(* IEC 61131-3 sources: programs/VI-54/VI-54_20171205/VI-54_20171205/Stations/Screen/LseClass170718/Class/CalcDeltaSC, 1 file *)

(* ---- CalcDeltaSC.st ---- *)
(*!
<Class
	Name               = "CalcDeltaSC"
	Revision           = "0.0"
	RealtimeTask       = "false"
	CyclicTask         = "false"
	BackgroundTask     = "false"
	Sigmatek           = "false"
	OSInterface        = "false"
	HighPriority       = "false"
	Automatic          = "false"
	UpdateMode         = "Prescan"
	SharedCommandTable = "true"
	Objectsize         = "(450,1320)">
	<Channels>
		<Server Name="OffsetZ" Visualized="false" Initialize="false" WriteProtected="false" Retentive="false"/>
	</Channels>
	<Network Name="CalcDeltaSC">
		<!-- List of Components in this network -->
		<Components>
			<Object
				Name       = "_base"
				Class      = "CalcDelta"
				Position   = "(218,120)"
				Visualized = "true"
				Remotely   = "true">
				<Channels>
					<Server Name="ActPos1"/>
					<Server Name="ActPos2"/>
					<Server Name="ActPos3"/>
					<Server Name="ActPos4"/>
					<Server Name="ClassSvr"/>
					<Server Name="DragCalcDelay" Value="0"/>
					<Server Name="HeadRadius" Value="500000"/>
					<Server Name="MotorArm" Value="3200000"/>
					<Server Name="MotorRadius" Value="2000000"/>
					<Server Name="RobotArm" Value="8500000"/>
					<Server Name="RobotRotAxisZ"/>
					<Server Name="SetPos1_Control"/>
					<Server Name="SetPos2_Control"/>
					<Server Name="SetPos3_Control"/>
					<Server Name="SetPos4_Control"/>
					<Server Name="XW1"/>
					<Server Name="XW2"/>
					<Server Name="XW3"/>
					<Server Name="XW4"/>
					<Client Name="Ax101"/>
					<Client Name="Ax102"/>
					<Client Name="Ax103"/>
					<Client Name="Ax104"/>
				</Channels>
			</Object>
		</Components>
		<Comments>
		</Comments>
		<!-- List of Connections in this network -->
		<Connections>
			<Connection Source="this.ClassSvr" Destination="_base.ClassSvr" Vertices="(946,210),(774,210),"/>
			<Connection Source="this.ActPos1" Destination="_base.ActPos1" Vertices="(946,270),(774,270),"/>
			<Connection Source="this.SetPos1_Control" Destination="_base.SetPos1_Control" Vertices="(946,330),(774,330),"/>
			<Connection Source="this.XW1" Destination="_base.XW1" Vertices="(946,390),(774,390),"/>
			<Connection Source="this.ActPos2" Destination="_base.ActPos2" Vertices="(946,450),(774,450),"/>
			<Connection Source="this.SetPos2_Control" Destination="_base.SetPos2_Control" Vertices="(946,510),(774,510),"/>
			<Connection Source="this.XW2" Destination="_base.XW2" Vertices="(946,570),(774,570),"/>
			<Connection Source="this.ActPos3" Destination="_base.ActPos3" Vertices="(946,630),(774,630),"/>
			<Connection Source="this.SetPos3_Control" Destination="_base.SetPos3_Control" Vertices="(946,690),(774,690),"/>
			<Connection Source="this.XW3" Destination="_base.XW3" Vertices="(946,750),(774,750),"/>
			<Connection Source="this.ActPos4" Destination="_base.ActPos4" Vertices="(946,810),(774,810),"/>
			<Connection Source="this.SetPos4_Control" Destination="_base.SetPos4_Control" Vertices="(946,870),(774,870),"/>
			<Connection Source="this.XW4" Destination="_base.XW4" Vertices="(946,930),(774,930),"/>
			<Connection Source="this.DragCalcDelay" Destination="_base.DragCalcDelay" Vertices="(946,990),(774,990),"/>
			<Connection Source="this.HeadRadius" Destination="_base.HeadRadius" Vertices="(946,1050),(774,1050),"/>
			<Connection Source="this.MotorRadius" Destination="_base.MotorRadius" Vertices="(946,1110),(774,1110),"/>
			<Connection Source="this.RobotArm" Destination="_base.RobotArm" Vertices="(946,1170),(774,1170),"/>
			<Connection Source="this.MotorArm" Destination="_base.MotorArm" Vertices="(946,1230),(774,1230),"/>
			<Connection Source="this.RobotRotAxisZ" Destination="_base.RobotRotAxisZ" Vertices="(946,1290),(774,1290),"/>
			<Connection Source="_base.Ax101" Destination="this.Ax101" Vertices="(218,210),(38,210),"/>
			<Connection Source="_base.Ax102" Destination="this.Ax102" Vertices="(218,270),(38,270),"/>
			<Connection Source="_base.Ax103" Destination="this.Ax103" Vertices="(218,330),(38,330),"/>
			<Connection Source="_base.Ax104" Destination="this.Ax104" Vertices="(218,390),(38,390),"/>
		</Connections>
		<!-- Headerfiles -->
		<Options>
		</Options>
	</Network>
</Class>
*)
#pragma using CalcDelta

CalcDeltaSC : CLASS
: CalcDelta
  //Servers:
	OffsetZ 	: SvrCh_DINT;
  //Clients:
  //Variables:
  //Functions:
				//! <Function Comment="Solves the direct kinematic problem:&#13;&#10;computes the effector-position and -orientation [world-coordinates] from the motor positions [ApplicationUnits]" Name="User_CalcDirectKinematic"/>
	FUNCTION VIRTUAL GLOBAL User_CalcDirectKinematic
		VAR_INPUT
			pMotorPos 	: ^_LMCPROF_POS;			//! <Variable Comment="pointer to the motor positions [ApplicationUnits] (input)" Name="User_CalcDirectKinematic.pMotorPos"/>
			pEffectorPos 	: ^_LMCPROF_POS;			//! <Variable Comment="pointer to the effector positions and -angles [world-coordinates] (output)" Name="User_CalcDirectKinematic.pEffectorPos"/>
		END_VAR
		VAR_OUTPUT
			ErrorNo 	: DINT;			//! <Variable Comment=" 0 ... no error&#13;&#10;&gt;0 ... errorcode" Name="User_CalcDirectKinematic.ErrorNo"/>
		END_VAR;
				//! <Function Comment="Solves the inverse kinematic problem:&#13;&#10;computes the motor positions [ApplicationUnits] from the effector-position and -orientation [world-coordinates]" Name="User_CalcInverseKinematic"/>
	FUNCTION VIRTUAL GLOBAL User_CalcInverseKinematic
		VAR_INPUT
			pEffectorPos 	: ^_LMCPROF_POS;			//! <Variable Comment="pointer to the effector positions and -angles [world-coordinates] (inpüt)" Name="User_CalcInverseKinematic.pEffectorPos"/>
			pMotorPos 	: ^_LMCPROF_POS;			//! <Variable Comment="pointer to the motor positions [ApplicationUnits] (output)" Name="User_CalcInverseKinematic.pMotorPos"/>
		END_VAR
		VAR_OUTPUT
			ErrorNo 	: DINT;			//! <Variable Comment=" 0 ... no error&#13;&#10;&gt;0 ... errorcode" Name="User_CalcInverseKinematic.ErrorNo"/>
		END_VAR;
  //Tables:
	FUNCTION @STD
		VAR_OUTPUT
			ret_code	: CONFSTATES;
		END_VAR;
	FUNCTION GLOBAL TAB @CT_;
END_CLASS;

FUNCTION VIRTUAL GLOBAL CalcDeltaSC::User_CalcDirectKinematic
	VAR_INPUT
		pMotorPos 	: ^_LMCPROF_POS;
		pEffectorPos 	: ^_LMCPROF_POS;
	END_VAR
	VAR_OUTPUT
		ErrorNo 	: DINT;
	END_VAR

  ErrorNo := CalcDelta::User_CalcDirectKinematic(pMotorPos, pEffectorPos);
  pEffectorPos^.Pos3 += OffsetZ;

END_FUNCTION

FUNCTION VIRTUAL GLOBAL CalcDeltaSC::User_CalcInverseKinematic
	VAR_INPUT
		pEffectorPos 	: ^_LMCPROF_POS;
		pMotorPos 	: ^_LMCPROF_POS;
	END_VAR
	VAR_OUTPUT
		ErrorNo 	: DINT;
	END_VAR

  pEffectorPos^.Pos3 -= OffsetZ;
  ErrorNo := CalcDelta::User_CalcInverseKinematic(pEffectorPos, pMotorPos);

END_FUNCTION
